(* IEC 61131-3 sources: volt/packages/volt-lsp-iec/test-corpus/awa-palletizer/Device/Plc Logic/Application, 2 files *)

(* ---- GVL_ComponentHardware.gvl ---- *)
(* This code is generated automatically *)
(* Don't change the content! *)

{attribute 'qualified_only'}
{attribute 'linkalways'}
VAR_GLOBAL
	//Controller
	Device 	: L_IC1P_ComponentHardware;

END_VAR

(* ---- GVL_ComponentHardwareCall.pou ---- *)
{attribute 'linkalways'}
PROGRAM GVL_ComponentHardwareCall
VAR
END_VAR
%LANGUAGE ST
(* This code is generated automatically *)
(* Don't change the content! *)

//Controller
GVL_ComponentHardware.Device();

END_PROGRAM
